// 40 Visualizations/BACNET_PARAMETER/VIS_DIA_BACNET_PARAMETER
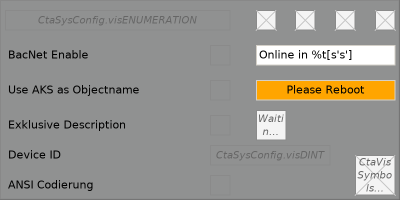
VISUALIZATION VIS_DIA_BACNET_PARAMETER  // 400x200
VAR_INPUT
	ITF_BACNET_PARAMETER_IN : ITF_BACNET_PARAMETER;
END_VAR
    Rectangle (0,0 400x200)
    Label (5,40 200x30), "BacNet Enable"
    Frame (210,45 20x20)
        shows CtaSysConfig.visBOOL(visfbBOOLIn := ITF_BACNET_PARAMETER_IN.P_fbxEnableBacNet)
    Label (5,75 200x30), "Use AKS as Objectname"
    Frame (210,80 20x20)
        shows CtaSysConfig.visBOOL(visfbBOOLIn := ITF_BACNET_PARAMETER_IN.P_fbxUseAKS)
    Frame (5,10 225x20), text list: 'KBOB_REV_TXT', text index: CtaSysConfig.fcGetEnumerationId(GVL_BACNET.fbBacNetParameter.fbenBacNetKbobRev)
        shows CtaSysConfig.visENUMERATION(visfbENUIn := ITF_BACNET_PARAMETER_IN.P_fbenBacNetKbobRev)
    Label (5,110 200x30), "Exklusive Description"
    Frame (210,115 20x20)
        shows CtaSysConfig.visBOOL(visfbBOOLIn := ITF_BACNET_PARAMETER_IN.P_fbxUseExklTxtList)
    Textfield (256,45 139x20), "Online in %t[s's']", text variable: ITF_BACNET_PARAMETER_IN.proTimeToOnline, invisible if: ITF_BACNET_PARAMETER_IN.proTimeToOnline = T#0s OR NOT ITF_BACNET_PARAMETER_IN.P_fbxEnableBacNet.proValue
    Image (335,10 20x20), invisible if: ITF_BACNET_PARAMETER_IN.proTimeToOnline = T#0s, image: CtaVisSymbols.ImagePool.Hourglass
    Image (375,10 20x20), invisible if: NOT ITF_BACNET_PARAMETER_IN.proCreate OR ITF_BACNET_PARAMETER_IN.proRebootRequired OR ITF_BACNET_PARAMETER_IN.proTimeToOnline <> T#0s, image: CtaVisSymbols.ImagePool.check_green
    Image (295,10 20x20), invisible if: NOT ITF_BACNET_PARAMETER_IN.proDelete OR ITF_BACNET_PARAMETER_IN.proTimeToOnline <> T#0s, image: CtaVisSymbols.ImagePool.close_red
    Image (256,10 20x20), invisible if: ITF_BACNET_PARAMETER_IN.proTimeToOnline <> T#0s OR NOT ITF_BACNET_PARAMETER_IN.proRebootRequired, image: CtaVisSymbols.ImagePool.refresh_solo_black
    Textfield (256,80 139x20), "Please Reboot", invisible if: ITF_BACNET_PARAMETER_IN.proTimeToOnline <> T#0s OR NOT ITF_BACNET_PARAMETER_IN.proRebootRequired
    Frame (210,145 120x20)
        shows CtaSysConfig.visDINT(visfbDINTIn := ITF_BACNET_PARAMETER_IN.P_fbdiDeviceId)
    Label (5,140 200x30), "Device ID"
    Image (355,155 40x40), image: CtaVisSymbols.ImagePool.database_black
        OnMouseClick:  Dialog=DIA_BACNET_LIST, OpenModal=True, OpenCentered=True
    Frame (210,175 20x20)
        shows CtaSysConfig.visBOOL(visfbBOOLIn := ITF_BACNET_PARAMETER_IN.P_fbxAnsiCodiert)
    Label (5,170 200x30), "ANSI Codierung"
    WaitingSymbolCube (256,110 30x30), invisible if: ITF_BACNET_PARAMETER_IN.proTimeToOnline = T#0s OR NOT ITF_BACNET_PARAMETER_IN.P_fbxEnableBacNet.proValue
END_VISUALIZATION

// 40 Visualizations/BACNET_PARAMETER/VIS_BACNET_APP
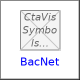
VISUALIZATION VIS_BACNET_APP  // 80x80
    Image (20,10 40x40), image: CtaVisSymbols.ImagePool.lan
    Label (15,47 50x30), "BacNet"
    RoundedRectangle (0,0 80x80)
        OnMouseClick:  Dialog=DIA_BACNET_PARAMETER, Parameters={ITF_BACNET_PARAMETER_IN: GVL_BACNET.fbBacNetParameter}, OpenCentered=True
END_VISUALIZATION

// 40 Visualizations/BACNET_PARAMETER/DIA_BACNET_LIST
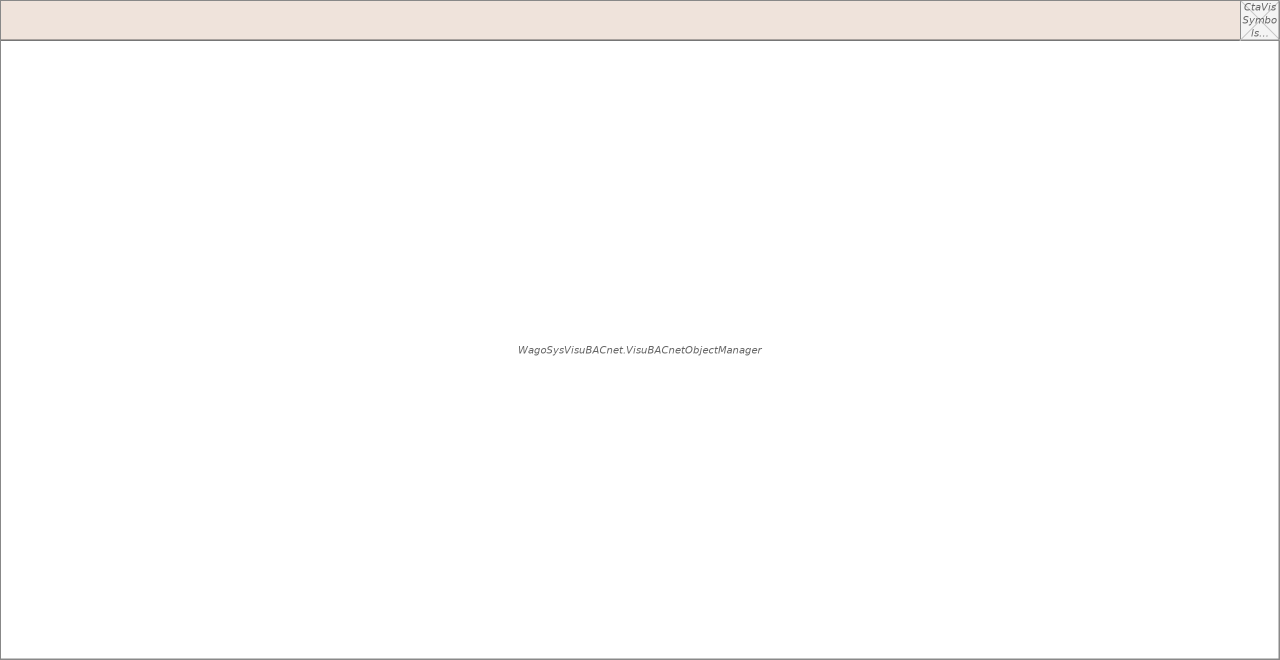
VISUALIZATION DIA_BACNET_LIST  // 1280x660
    Frame (0,40 1280x620)
        shows WagoSysVisuBACnet.VisuBACnetObjectManager()
    Rectangle (0,0 1280x40)
    Image (1240,0 40x40), image: CtaVisSymbols.ImagePool.close_solo_black
        OnMouseClick:  Dialog=DIA_BACNET_LIST, Result=OK, NumpadKeypadSet=True
END_VISUALIZATION

(* text list TXT_AT_ANTRIEB_STETIG_ENDING (id | default)
  A_BO_1 | _A_BO_1
  B_TL_1 | _B_TL_1
  C_EE_1 | _C_EE_1
  D_BV_1 | _D_BV_1
  E_BV_2 | _E_BV_2
  F_BI_1 | _F_BI_1
  G_AO_1 | _G_AO_1
  I_AI_1 | _I_AI_1
  K_BI_2 | _K_BI_2
  L_BV_3 | _L_BV_3
  H_TL_2 | _H_TL_2
  J_TL_3 | _J_TL_3
   |  *)

(* text list TXT_AT_ANTRIEB_STETIG_DESCRIPTION (id | default)
  A_BO_1 | Schaltbefehl
  B_TL_1 | Aufzeichnung Betriebsrückmeldung
  C_EE_1 | Instandhaltungsmeldung
  D_BV_1 | Betriebsdauer
  E_BV_2 | Handbetrieb
  F_BI_1 | Revisionsschalter
  G_AO_1 | Sollwertvorgabe
  I_AI_1 | Istwert
  K_BI_2 | CosPhi
  L_BV_3 | Störung
  H_TL_2 | Aufzeichnunng Sollwertvorgabe
  J_TL_3 | Aufzeichnung Istwert
   |  *)

(* text list TXT_AT_ANTRIEB_STETIG_PRESV (id | default)
  A_BO_1_ST_ACTIVE | 
  A_BO_1_ST_INACTIVE | 
  D_BV_1_ST_ACTIVE | 
  D_BV_1_ST_INACTIVE | 
   |  *)

(* text list TXT_AT_ANTRIEB_STETIG_EVENTMESSAGE (id | default)
  A_MV_1_ToOffNormal | ToOffNormal
  A_MV_1_ToFault | ToFault
  A_MV_1_ToNormal | ToNormal
  B_MI_1_ToOffNormal | ToOffNormal
  B_MI_1_ToFault | ToFault
  B_MI_1_ToNormal | ToNormal
  C_BV_1_ToOffNormal | ToOffNormal
  C_BV_1_ToFault | ToFault
  C_BV_1_ToNormal | ToNormal
  D_SC_1_ToOffNormal | ToOffNormal
  D_SC_1_ToFault | ToFault
  D_SC_1_ToNormal | ToNormal
   |  *)

(* text list TXT_AT_ANLAGENSCHALTER_NC (id | default)
  C_BV_1_NC | 128
  C_BV_1_ALV | TRUE
   |  *)

(* text list TXT_AT_ANLAGENSCHALTER_ENDING (id | default)
  A_MV_1 | _A_MV_1
  B_MI_1 | _B_MI_1
  C_BV_1 | _C_BV_1
  D_SC_1 | _D_SC_1
   |  *)

(* text list TXT_AT_ANLAGENSCHALTER_EVENTMESSAGE (id | default)
  A_MV_1_ToOffNormal | ToOffNormal
  A_MV_1_ToFault | ToFault
  A_MV_1_ToNormal | ToNormal
  B_MI_1_ToOffNormal | ToOffNormal
  B_MI_1_ToFault | ToFault
  B_MI_1_ToNormal | ToNormal
  C_BV_1_ToOffNormal | ToOffNormal
  C_BV_1_ToFault | ToFault
  C_BV_1_ToNormal | ToNormal
  D_SC_1_ToOffNormal | ToOffNormal
  D_SC_1_ToFault | ToFault
  D_SC_1_ToNormal | ToNormal
   |  *)

(* text list TXT_AT_ANLAGENSCHALTER_PRESV (id | default)
  A_MV_1_ST_1 | Aus
  A_MV_1_ST_2 | Ein
  B_MI_1_ST_1 | Auto
  B_MI_1_ST_2 | Aus
  B_MI_1_ST_3 | Ein
  C_BV_1_ST_INACTIVE | Auto
  C_BV_1_ST_ACTIVE | Hand
   |  *)

(* text list TXT_AT_ANTRIEB_STETIG_NC (id | default)
  A_BO_1_NC | 224
  B_TL_1_NC | 192
  C_EE_1_NC | 128
  E_BV_2_NC | 160
  E_BV_2_ALV | TRUE
  F_BI_1_ALV | FALSE
  F_BI_1_NC | 160
  I_AI_1_NC | 224
  K_BI_2_ALV | TRUE
  K_BI_2_NC | 96
  L_BV_3_ALV | TRUE
  L_BV_3_NC | 96
  H_TL_2 | 192
  J_TL_3 | 192
   |  *)

(* text list TXT_AT_ANLAGENSCHALTER_DESCRIPTION (id | default)
  A_MV_1 | Betriebswahl
  B_MI_1 | Betriebswahl Lokal
  C_BV_1 | Handbetrieb Nicht Auto
  D_SC_1 | Zeitschaltuhr
   |  *)

(* text list TXT_AT_MESSWERTGEBER_BINAR_DESCRIPTION (id | default)
  A_BI_1 | Istwert
  B_TL_1 | Trendlog
  C_BV_1 | Fehler
   |  *)

(* text list TXT_AT_MESSWERTGEBER_BINAR_ENDING (id | default)
  A_BI_1 | _A_BI_1
  B_TL_1 | _B_TL_1
  C_BV_1 | _C_BV_1
   |  *)

(* text list TXT_AT_MESSWERTGEBER_BINAR_NC (id | default)
  A_BI_1_NC | 224
  B_TL_1_NC | 192
  C_BV_1_NC | 96
  C_BV_1_ALV | TRUE
   |  *)

(* text list TXT_AT_MESSWERTGEBER_BINAR_EVENTMESSAGE (id | default)
  A_BI_1_ToOffNormal | ToOffNormal
  A_BI_1_1_ToFault | ToFault
  A_BI_1_1_ToNormal | ToNormal
  B_TL_1_ToOffNormal | ToOffNormal
  B_TL_1_ToFault | ToFault
  B_TL_1_ToNormal | ToNormal
  C_BV_1_ToOffNormal | ToOffNormal
  C_BV_1_ToFault | ToFault
  C_BV_1_ToNormal | ToNormal
   |  *)

(* text list TXT_AT_MESSWERTGEBER_BINAR_PRESV (id | default)
  A_BI_1_ST_ACTIVE | Ausgelöst
  A_BI_1_ST_INACTIVE | Normal
  C_BV_1_ST_ACTIVE | Ausgelöst
  C_BV_1_ST_INACTIVE | Normal
   |  *)

(* text list TXT_AT_MESSWERTGEBER_STETIG_NC (id | default)
  A_AI_1_NC | 224
  C_TL_1_NC | 192
  B_EE_1_NC | 96
   |  *)

(* text list TXT_AT_MESSWERTGEBER_STETIG_DESCRIPTION (id | default)
  A_AI_1 | Istwert
  C_TL_1 | Trendlog
  B_EE_1 | Voralarm
   |  *)

(* text list TXT_AT_MESSWERTGEBER_STETIG_ENDING (id | default)
  A_AI_1 | _A_AI_1
  C_TL_1 | _B_TL_1
  B_EE_1 | _C_EE_1
   |  *)

(* text list TXT_AT_MESSWERTGEBER_STETIG_EVENTMESSAGE (id | default)
  A_AI_1_ToOffNormal | ToOffNormal
  A_AI_1_ToFault | ToFault
  A_AI_1_ToNormal | ToNormal
  C_TL_1_ToOffNormal | ToOffNormal
  C_TL_1_ToFault | ToFault
  C_TL_1_ToNormal | ToNormal
  B_EE_1_ToOffNormal | ToOffNormal
  B_EE_1_ToFault | ToFault
  B_EE_1_ToNormal | ToNormal
   |  *)

(* text list TXT_AT_MESSWERTGEBER_STETIG_PRESV (id | default)
   |  *)

(* text list KBOB_REV_TXT (id | default)
  0 | KBOB REV2017 V1
  1 | KBOB REV2021 V2
   |  *)

(* text list TXT_AT_AUTOMATIONSSTATION_DESCRIPTION (id | default)
  A_DV_1 | CTA-Anlage
  B_CL_1 | Kalender variable Feiertage
  C_CL_2 | Kalender halbe Tage
  D_CL_3 | Kalender feste Feiertage
  E_CL_4 | Kalender Ferien
  F_EL_1 | Eventlog
  G_NC_1 | Sicherheitsalarm NC 1
  G_NC_2 | Sicherheitsalarm NC 2
  G_NC_3 | Sicherheitsalarm NC 3
  G_NC_4 | Sicherheitsalarm NC 4
  H_NC_32 | Objektschutz NC 32
  H_NC_33 | Objektschutz NC 33
  H_NC_34 | Objektschutz NC 34
  H_NC_35 | Objektschutz NC 35
  I_NC_64 | Technischer Alarm NC 64
  I_NC_65 | Technischer Alarm NC 65
  I_NC_66 | Technischer Alarm NC 66
  I_NC_67 | Technischer Alarm NC 67
  J_NC_96 | Technische Störung NC 96
  J_NC_97 | Technische Störung NC 97
  J_NC_98 | Technische Störung NC 98
  J_NC_99 | Technische Störung NC 99
  K_NC_128 | Präventive Wartungsmeldung NC 128
  K_NC_129 | Präventive Wartungsmeldung NC 129
  K_NC_130 | Präventive Wartungsmeldung NC 130
  K_NC_131 | Präventive Wartungsmeldung NC 131
  L_NC_160 | Revisionsmeldung NC 160
  L_NC_161 | Revisionsmeldung NC 161
  L_NC_162 | Revisionsmeldung NC 162
  L_NC_163 | Revisionsmeldung NC 163
  M_NC_192 | Trenddaten NC 192
  M_NC_193 | Trenddaten NC 193
  N_NC_224 | Betriebs - oder Statusmeldung NC 224
  N_NC_225 | Betriebs - oder Statusmeldung NC 225
  O_BV_1 | CPU Status
  P_BV_2 | I/O Modul Status
  Q_BV_3 | Meldung Handeingriff I/O Modul
  R_BV_4 | Heartbeat
  S_BV_5 | BacNet Stack Status
   |  *)

(* text list TXT_AT_AUTOMATIONSSTATION_ENDING (id | default)
  A_DV_1 | _A_DV_1
  B_CL_1 | _B_CL_1
  C_CL_2 | _C_CL_2
  D_CL_3 | _D_CL_3
  E_CL_4 | _E_CL_4
  F_EL_1 | _F_EL_1
  G_NC_1 | _G_NC_1
  G_NC_2 | _G_NC_2
  G_NC_3 | _G_NC_3
  G_NC_4 | _G_NC_4
  H_NC_32 | _H_NC_32
  H_NC_33 | _H_NC_33
  H_NC_34 | _H_NC_34
  H_NC_35 | _H_NC_35
  I_NC_64 | _I_NC_64
  I_NC_65 | _I_NC_65
  I_NC_66 | _I_NC_66
  I_NC_67 | _I_NC_67
  J_NC_96 | _J_NC_96
  J_NC_97 | _J_NC_97
  J_NC_98 | _J_NC_98
  J_NC_99 | _J_NC_99
  K_NC_128 | _K_NC_128
  K_NC_129 | _K_NC_129
  K_NC_130 | _K_NC_130
  K_NC_131 | _K_NC_131
  L_NC_160 | _L_NC_160
  L_NC_161 | _L_NC_161
  L_NC_162 | _L_NC_162
  L_NC_163 | _L_NC_163
  M_NC_192 | _M_NC_192
  M_NC_193 | _M_NC_193
  N_NC_224 | _N_NC_224
  N_NC_225 | _N_NC_225
  O_BV_1 | _O_BV_1
  P_BV_2 | _P_BV_2
  Q_BV_3 | _Q_BV_3
  R_BV_4 | _R_BV_4
  S_BV_5 | _S_BV_5
   |  *)

(* text list TXT_AT_AUTOMATIONSSTATION_NC (id | default)
  O_BV_1_NC | 96
  O_BV_1_ALV | TRUE
  P_BV_2_NC | 96
  P_BV_2_ALV | TRUE
  Q_BV_3_NC | 128
  Q_BV_3_ALV | TRUE
  R_BV_4_NC | 224
  R_BV_4_ALV | TRUE
  S_BV_5_NC | 96
  S_BV_5_ALV | TRUE
   |  *)

(* text list TXT_AT_AUTOMATIONSSTATION_PRESV (id | default)
  O_BV_1_ST_ACTIVE | Fehler
  O_BV_1_ST_INACTIVE | Normal
  P_BV_2_ST_ACTIVE | Fehler
  P_BV_2_ST_INACTIVE | Normal
  Q_BV_3_ST_ACTIVE | Hand
  Q_BV_3_ST_INACTIVE | Normal
  R_BV_4_ST_ACTIVE | Ein
  R_BV_4_ST_INACTIVE | Aus
  S_BV_5_ST_ACTIVE | Fehler
  S_BV_5_ST_INACTIVE | Normal
   |  *)

(* text list TXT_AT_AUTOMATIONSSTATION_EVENTMESSAGE (id | default)
  O_BV_1_ToOffNormal | ToOffNormal
  O_BV_1_ToFault | ToFault
  O_BV_1_ToNormal | ToNormal
  P_BV_2_ToOffNormal | ToOffNormal
  P_BV_2_ToFault | ToFault
  P_BV_2_ToNormal | ToNormal
  Q_BV_3_ToOffNormal | ToOffNormal
  Q_BV_3_ToFault | ToFault
  Q_BV_3_ToNormal | ToNormal
  R_BV_4_ToOffNormal | ToOffNormal
  R_BV_4_ToFault | ToFault
  R_BV_4_ToNormal | ToNormal
  S_BV_5_ToOffNormal | ToOffNormal
  S_BV_5_ToFault | ToFault
  S_BV_5_ToNormal | ToNormal
   |  *)

(* text list TXT_AT_ANLAGEFUNKTION_DESCRIPTION (id | default)
  A_BV_1 | Sammelmeldung Objektschutz
  B_BV_2 | Sammelmeldung Technischer Alarm
  C_BV_3 | Sammelmeldung Technische Störung
  D_BV_4 | Sammelmeldung Wartungsmeldung
  E_BI_1 | Bedienung Lokal
  F_BV_5 | Alarmunterdrückung
  G_BO_1 | Signalisation Betrieb
  H_BO_2 | Signalisation Sammelalarm
  I_BO_3 | Signalisation Bedienung Lokal
  J_SC_1 | Zeitschaltuhr
   |  *)

(* text list TXT_AT_ANLAGEFUNKTION_ENDING (id | default)
  A_BV_1 | _A_BV_1
  B_BV_2 | _B_BV_2
  C_BV_3 | _C_BV_3
  D_BV_4 | _D_BV_4
  E_BI_1 | _E_BI_1
  F_BV_5 | _F_BV_5
  G_BO_1 | _G_BO_1
  H_BO_2 | _H_BO_2
  I_BO_3 | _I_BO_3
  J_SC_1 | _J_SC_1
   |  *)

(* text list TXT_AT_ANLAGEFUNKTION_EVENTMESSAGE (id | default)
  A_BV_1_ToOffNormal | ToOffNormal
  A_BV_1_ToFault | ToFault
  A_BV_1_ToNormal | ToNormal
  B_BV_2_ToOffNormal | ToOffNormal
  B_BV_2_ToFault | ToFault
  B_BV_2_ToNormal | ToNormal
  C_BV_3_ToOffNormal | ToOffNormal
  C_BV_3_ToFault | ToFault
  C_BV_3_ToNormal | ToNormal
  D_BV_4_ToOffNormal | ToOffNormal
  D_BV_4_ToFault | ToFault
  D_BV_4_ToNormal | ToNormal
  E_BI_1_ToOffNormal | ToOffNormal
  E_BI_1_ToFault | ToFault
  E_BI_1_ToNormal | ToNormal
  F_BV_5_ToOffNormal | ToOffNormal
  F_BV_5_ToFault | ToFault
  F_BV_5_ToNormal | ToNormal
  G_BO_1_ToOffNormal | ToOffNormal
  G_BO_1_ToFault | ToFault
  G_BO_1_ToNormal | ToNormal
  H_BO_2_ToOffNormal | ToOffNormal
  H_BO_2_ToFault | ToFault
  H_BO_2_ToNormal | ToNormal
  I_BO_3_ToOffNormal | ToOffNormal
  I_BO_3_ToFault | ToFault
  I_BO_3_ToNormal | ToNormal
  J_SC_1_ToOffNormal | ToOffNormal
  J_SC_1_ToFault | ToFault
  J_SC_1_ToNormal | ToNormal
   |  *)

(* text list TXT_AT_ANLAGEFUNKTION_NC (id | default)
  A_BV_1_NC | 96
  A_BV_1_ALV | TRUE
  B_BV_2_NC | 96
  B_BV_2_ALV | TRUE
  C_BV_3_NC | 96
  C_BV_3_ALV | TRUE
  D_BV_4_NC | 96
  D_BV_4_ALV | TRUE
  E_BI_1_NC | 96
  E_BI_1_ALV | TRUE
  F_BV_5_NC | 96
  F_BV_5_ALV | TRUE
   |  *)

(* text list TXT_AT_ANLAGEFUNKTION_PRESV (id | default)
  A_BV_1_ST_ACTIVE | Ausgelöst
  A_BV_1_ST_INACTIVE | Normal
  B_BV_2_ST_ACTIVE | Ausgelöst
  B_BV_2_ST_INACTIVE | Normal
  C_BV_3_ST_ACTIVE | Ausgelöst
  C_BV_3_ST_INACTIVE | Normal
  D_BV_4_ST_ACTIVE | Ausgelöst
  D_BV_4_ST_INACTIVE | Normal
  E_BI_1_ST_ACTIVE | Hand
  E_BI_1_ST_INACTIVE | Normal
  F_BV_5_ST_ACTIVE | Inaktiv
  F_BV_5_ST_INACTIVE | Aktive
  G_BO_1_ST_ACTIVE | Ein
  G_BO_1_ST_INACTIVE | Aus
  H_BO_2_ST_ACTIVE | Ein
  H_BO_2_ST_INACTIVE | Aus
  I_BO_3_ST_ACTIVE | Ein
  I_BO_3_ST_INACTIVE | Aus
   |  *)

(* text list TXT_AT_ZÄHLER_DESCRIPTION (id | default)
  A_AV_1 | Messwert
  B_TL_1 | Trendlog
  C_BV_1 | Fehler
   |  *)

(* text list TXT_AT_ZÄHLER_ENDING (id | default)
  A_AV_1 | _A_AV_1
  B_TL_1 | _B_TL_1
  C_BV_1 | _C_BV_1
   |  *)

(* text list TXT_AT_ZÄHLER_EVENTMESSAGE (id | default)
  A_AV_1_ToOffNormal | ToOffNormal
  A_AV_1_ToFault | ToFault
  A_AV_1_ToNormal | ToNormal
  B_TL_1_ToOffNormal | ToOffNormal
  B_TL_1_ToFault | ToFault
  B_TL_1_ToNormal | ToNormal
  C_BV_1_ToOffNormal | ToOffNormal
  C_BV_1_ToFault | ToFault
  C_BV_1_ToNormal | ToNormal
   |  *)

(* text list TXT_AT_ZÄHLER_NC (id | default)
  A_AV_1_NC | 224
  B_TL_1_NC | 192
  C_BV_1_NC | 96
  C_BV_1_ALV | TRUE
   |  *)

(* text list TXT_AT_ZÄHLER_PRESV (id | default)
  C_BV_1_ST_ACTIVE | Ausgelöst
  C_BV_1_ST_INACTIVE | Normal
   |  *)

(* text list TXT_AT_STELLORGAN_STETIG_ENDING (id | default)
  A_AO_1 | _A_AO_1
  B_AI_1 | _B_AI_1
  C_TL_1 | _C_TL_1
  D_BI_1 | _D_BI_1
  E_BI_2 | _E_BI_2
  F_BV_1 | _F_BV_1
   |  *)

(* text list TXT_AT_STELLORGAN_STETIG_EVENTMESSAGE (id | default)
  A_AO_1_ToOffNormal | ToOffNormal
  A_AO_1_ToFault | ToFault
  A_AO_1_ToNormal | ToNormal
  B_AI_1_ToOffNormal | ToOffNormal
  B_AI_1_ToFault | ToFault
  B_AI_1_ToNormal | ToNormal
  B_EE_1_ToOffNormal | ToOffNormal
  B_EE_1_ToFault | ToFault
  B_EE_1_ToNormal | ToNormal
  C_TL_1_ToOffNormal | ToOffNormal
  C_TL_1_ToFault | ToFault
  C_TL_1_ToNormal | ToNormal
  D_BI_1_ToOffNormal | ToOffNormal
  D_BI_1_ToFault | ToFault
  D_BI_1_ToNormal | ToNormal
  E_BI_2_ToOffNormal | ToOffNormal
  E_BI_2_ToFault | ToFault
  E_BI_2_ToNormal | ToNormal
  F_BV_1_ToOffNormal | ToOffNormal
  F_BV_1_ToFault | ToFault
  F_BV_1_ToNormal | ToNormal
   |  *)

(* text list TXT_AT_STELLORGAN_STETIG_DESCRIPTION (id | default)
  A_AO_1 | Stellwert
  B_AI_1 | Stellwertrückmeldung
  C_TL_1 | Aufzeichnung Stellwert
  D_BI_1 | Stellungsrückmeldung Zu
  E_BI_2 | Stellungsrückmeldung Auf
  F_BV_1 | Störung Stellorgan
   |  *)

(* text list TXT_AT_STELLORGAN_STETIG_NC (id | default)
  A_AO_1_NC | 96
  B_AI_1_NC | 96
  C_TL_1_NC | 96
  D_BI_1_NC | 96
  E_BI_2_NC | 96
  F_BV_1_NC | 96
  F_BV_1_ALV | TRUE
  E_BI_2_ALV | TRUE
  D_BI_1_ALV | TRUE
   |  *)

(* text list TXT_AT_STELLORGAN_STETIG_PRESV (id | default)
  D_BI_1_ST_ACTIVE | Zu
  D_BI_1_ST_INACTIVE | Inaktiv
  E_BI_2_ST_ACTIVE | Auf
  E_BI_2_ST_INACTIVE | Inaktiv
  F_BV_1_ST_ACTIVE | Störung
  F_BV_1_ST_INACTIVE | Normal
   |  *)
